{attribute 'GeneratedUsingTerminal: EK1122-0000-0018'}
{attribute addProperty BoxType "EK1122-0000-0018"}
{attribute addProperty Id "Beckhoff_EL15xxsub_EK1100EK1100_AB5A94672"}
{attribute addProperty CRC "3059104709"}
{attribute addProperty Size "2"}
TYPE Beckhoff_EL15xxEK1122_B6563BC5 EXTENDS EK1122_AB5A9467 :
STRUCT
	{attribute addProperty Name "Beckhoff_EL15xxsub_EK1100"}
	Beckhoff_EL15xxsub_EK1100 : EK1100_AB5A9467;
END_STRUCT
END_TYPE

(* stored: Version 1.2.0.0, ProductVersion 3.1.4024.9
   DUT Beckhoff_EL15xxEK1122_B6563BC5: Id {ed82fd91-328c-4ef2-aaea-f1019bb0330f} *)
